// TIA Portal V15 export
FUNCTION "Preset_main" : Void   // FC30, SCL
TITLE = Presethantering / Preset handling
{ S7_Optimized_Access := 'TRUE' }
VERSION : 0.1
// stored: AutoNumber true, IsIECCheckEnabled false, SetENOAutomatically False
   VAR_INPUT
      Set : Bool;
      Store : Bool;
      Index : Int;
   END_VAR
BEGIN
// Presethantering / Preset handling
END_FUNCTION
